// TIA Portal V16 export
// export: Created 2024-09-05T17:40:15.5377235Z, ExportSetting WithDefaults, DisplayName Totally Integrated Automation Portal, DisplayVersion V16 Update 6, DisplayName TIA Portal Version Control Interface, DisplayVersion V16 Update 2, DisplayName TIA Portal Openness, DisplayVersion V16 Update 6, DisplayName STEP 7 Professional, DisplayVersion V16 Update 6, DisplayName STEP 7 Safety, DisplayVersion V16, DisplayName WinCC Advanced, DisplayVersion V16 Update 6
TYPE "MII_Interface.MII_METHODS.M001_GET_LOCAL_TIME.Outputs"
// stored: IsFailsafeCompliant false
   STRUCT
      DATETIME_LOCAL { ExternalAccessible := 'False'; ExternalVisible := 'False'; ExternalWritable := 'False'} : LDT;
      DATE_TIME_UTC { ExternalAccessible := 'False'; ExternalVisible := 'False'; ExternalWritable := 'False'} : LDT;
   END_STRUCT;
END_TYPE
